TYPE ST_AutoMode_ReloadRoundBeltBox :
STRUCT
	Command : ST_ReloadRoundBelt_Ctrl;
	Status : ST_ReloadRoundBelt_Status;
	Info : ST_ReloadRoundBeltBox_Info;
	AClampMoveDone	: BOOL;
	BClampMoveDone	: BOOL;
END_STRUCT
END_TYPE

(* stored: Version 1.1.0.1, ProductVersion 3.1.4024.13
   DUT ST_AutoMode_ReloadRoundBeltBox: Id {c1efc38b-8a16-4b97-8f78-ae904abb897d} *)
